// TIA Portal V20 export
FUNCTION_BLOCK "Conveyor_C4"   // FB10025, LAD
// stored: MemoryReserve 100, Namespace Conveyor4, SetENOAutomatically false
   VAR
      statManRight : Bool;
      statManLeft : Bool;
      statAutoRight : Bool;
      statAutoLeft : Bool;
      statRunning : Bool;
      reLightBarrier { S7_SetPoint := 'True'} : R_TRIG;
      tonDelayStart { S7_SetPoint := 'True'} : TON_TIME;
   END_VAR
   VAR_TEMP
      tmpHorn : Bool;
   END_VAR
BEGIN

REGION Network 1: Manual - Run conveyor LEFT
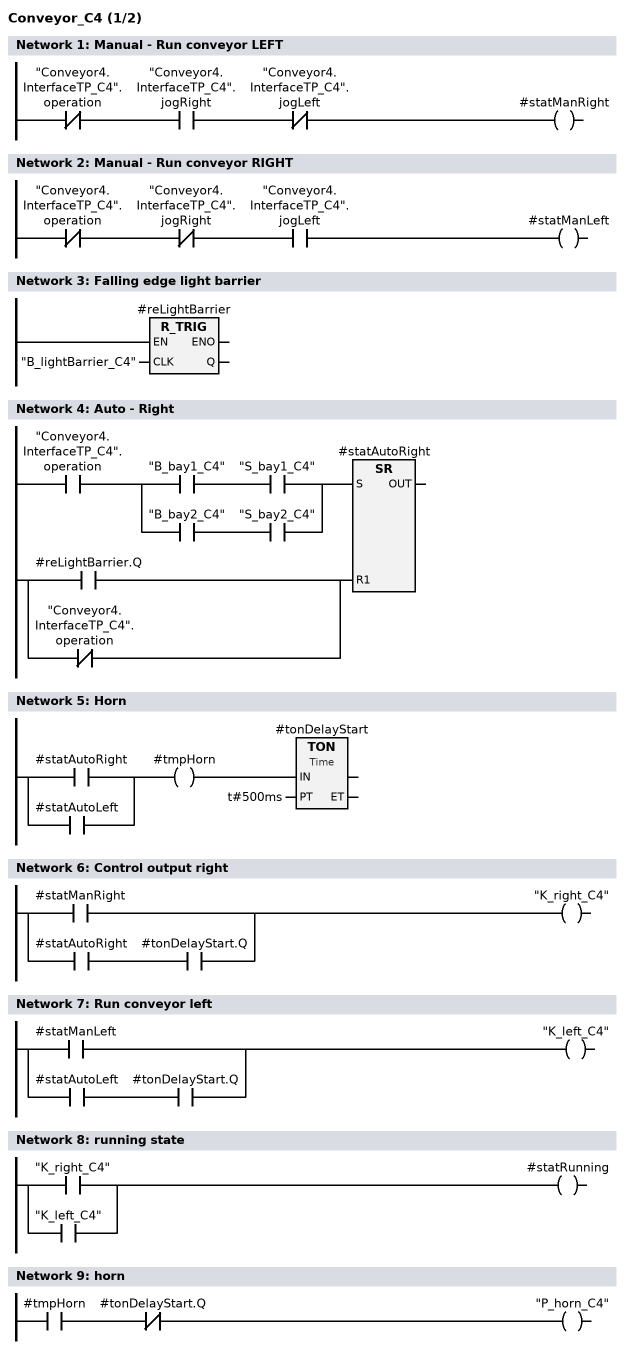
   RUNG wire#powerrail
      I_Contact( "Conveyor4.InterfaceTP_C4".operation )
      Contact( "Conveyor4.InterfaceTP_C4".jogRight )
      I_Contact( "Conveyor4.InterfaceTP_C4".jogLeft )
      Coil( #statManRight )
   END_RUNG
   // the same network as SCL:
   #statManRight := NOT "Conveyor4.InterfaceTP_C4".operation AND "Conveyor4.InterfaceTP_C4".jogRight AND NOT "Conveyor4.InterfaceTP_C4".jogLeft;
END_REGION

REGION Network 2: Manual - Run conveyor RIGHT
   RUNG wire#powerrail
      I_Contact( "Conveyor4.InterfaceTP_C4".operation )
      I_Contact( "Conveyor4.InterfaceTP_C4".jogRight )
      Contact( "Conveyor4.InterfaceTP_C4".jogLeft )
      Coil( #statManLeft )
   END_RUNG
   // the same network as SCL:
   #statManLeft := NOT "Conveyor4.InterfaceTP_C4".operation AND NOT "Conveyor4.InterfaceTP_C4".jogRight AND "Conveyor4.InterfaceTP_C4".jogLeft;
END_REGION

REGION Network 3: Falling edge light barrier
   RUNG wire#powerrail
      #reLightBarrier.R_TRIG(CLK := "B_lightBarrier_C4", Q =>)
   END_RUNG
   // the same network as SCL:
   #reLightBarrier(CLK := "B_lightBarrier_C4");   // R_TRIG
END_REGION

REGION Network 4: Auto - Right
   RUNG wire#powerrail
      Contact( "Conveyor4.InterfaceTP_C4".operation )
      wire#w1
      Contact( "B_bay1_C4" )
      Contact( "S_bay1_C4" )
      wire#w2
      S_SR(operand := #statAutoRight, r1 := wire#w3)
   END_RUNG
   RUNG wire#w1
      Contact( "B_bay2_C4" )
      Contact( "S_bay2_C4" )
   END_RUNG wire#w2
   RUNG wire#powerrail
      Contact( #reLightBarrier.Q )
   END_RUNG wire#w3
   RUNG wire#powerrail
      I_Contact( "Conveyor4.InterfaceTP_C4".operation )
   END_RUNG wire#w3
   // the same network as SCL:
   IF "Conveyor4.InterfaceTP_C4".operation AND (("B_bay1_C4" AND "S_bay1_C4") OR ("B_bay2_C4" AND "S_bay2_C4")) THEN
       #statAutoRight := TRUE;   // SR flip-flop
   END_IF;
   IF #reLightBarrier.Q OR NOT "Conveyor4.InterfaceTP_C4".operation THEN #statAutoRight := FALSE; END_IF;
END_REGION

REGION Network 5: Horn
   RUNG wire#powerrail
      Contact( #statAutoRight )
      wire#w1
      Coil( #tmpHorn )
      { S7_Templates := "time_type := Time" } #tonDelayStart.TON(pt := t#500ms, et =>)
   END_RUNG
   RUNG wire#powerrail
      Contact( #statAutoLeft )
   END_RUNG wire#w1
   // the same network as SCL:
   #tmpHorn := #statAutoRight OR #statAutoLeft;
   #tonDelayStart(IN := #tmpHorn, PT := t#500ms);   // TON
END_REGION

REGION Network 6: Control output right
   RUNG wire#powerrail
      Contact( #statManRight )
      wire#w1
      Coil( "K_right_C4" )
   END_RUNG
   RUNG wire#powerrail
      Contact( #statAutoRight )
      Contact( #tonDelayStart.Q )
   END_RUNG wire#w1
   // the same network as SCL:
   "K_right_C4" := #statManRight OR (#statAutoRight AND #tonDelayStart.Q);
END_REGION

REGION Network 7: Run conveyor left
   RUNG wire#powerrail
      Contact( #statManLeft )
      wire#w1
      Coil( "K_left_C4" )
   END_RUNG
   RUNG wire#powerrail
      Contact( #statAutoLeft )
      Contact( #tonDelayStart.Q )
   END_RUNG wire#w1
   // the same network as SCL:
   "K_left_C4" := #statManLeft OR (#statAutoLeft AND #tonDelayStart.Q);
END_REGION

REGION Network 8: running state
   RUNG wire#powerrail
      Contact( "K_right_C4" )
      wire#w1
      Coil( #statRunning )
   END_RUNG
   RUNG wire#powerrail
      Contact( "K_left_C4" )
   END_RUNG wire#w1
   // the same network as SCL:
   #statRunning := "K_right_C4" OR "K_left_C4";
END_REGION

REGION Network 9: horn
   RUNG wire#powerrail
      Contact( #tmpHorn )
      I_Contact( #tonDelayStart.Q )
      Coil( "P_horn_C4" )
   END_RUNG
   // the same network as SCL:
   "P_horn_C4" := #tmpHorn AND NOT #tonDelayStart.Q;
END_REGION

REGION Network 10: indicator light bay 1
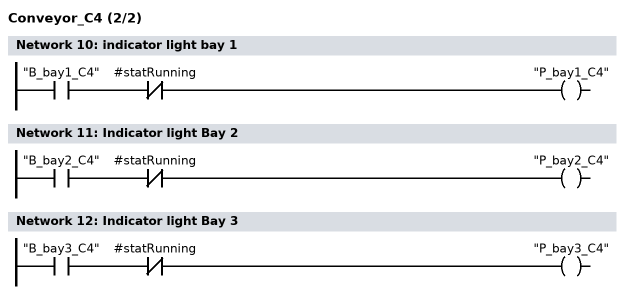
   RUNG wire#powerrail
      Contact( "B_bay1_C4" )
      I_Contact( #statRunning )
      Coil( "P_bay1_C4" )
   END_RUNG
   // the same network as SCL:
   "P_bay1_C4" := "B_bay1_C4" AND NOT #statRunning;
END_REGION

REGION Network 11: Indicator light Bay 2
   RUNG wire#powerrail
      Contact( "B_bay2_C4" )
      I_Contact( #statRunning )
      Coil( "P_bay2_C4" )
   END_RUNG
   // the same network as SCL:
   "P_bay2_C4" := "B_bay2_C4" AND NOT #statRunning;
END_REGION

REGION Network 12: Indicator light Bay 3
   RUNG wire#powerrail
      Contact( "B_bay3_C4" )
      I_Contact( #statRunning )
      Coil( "P_bay3_C4" )
   END_RUNG
   // the same network as SCL:
   "P_bay3_C4" := "B_bay3_C4" AND NOT #statRunning;
END_REGION
END_FUNCTION_BLOCK
